SUBAPPLICATION Uebung_039a_AX (* Spiegelabfolge V2 mit Schrittkette *)
  (* Standard: 61499-2; Description: Copyright (c) 2023 Meisterschulen am Ostbahnhof This program and the accompanying materials are made available under the terms of the Eclipse Public License 2.0 which is available at https://www.eclipse.org/legal/epl-2.0/ SPDX-License-Identifier: EPL-2.0 *)
  (* Version 1.0, 2023-10-23, Franz Höpfinger, Meisterschulen am Ostbahnhof, initial API and implementation and/or initial documentation *)
  PACKAGE Uebungen;
  IMPORT isobus::UT::io::Softkey::SoftKeyActivationCode::SK_RELEASED;
  IMPORT Uebungen::const::UT::DefaultPool::SoftKey_F1;
  IMPORT Uebungen::const::UT::DefaultPool::SoftKey_F2;
  IMPORT Uebungen::const::UT::DefaultPool::SoftKey_F8;
  IMPORT Uebungen::const::UT::DefaultPool::OutputNumber_N1;
  IMPORT logiBUS::io::DI::logiBUS_DI::Input_I1;
  IMPORT logiBUS::io::DI::logiBUS_DI::Input_I2;
  IMPORT logiBUS::io::DI::logiBUS_DI::Input_I3;
  IMPORT logiBUS::io::DI::logiBUS_DI::Input_I4;
  IMPORT logiBUS::io::DI::logiBUS_DI_Events::BUTTON_SINGLE_CLICK;
  IMPORT logiBUS::io::DQ::logiBUS_DO::Output_Q1;
  IMPORT logiBUS::io::DQ::logiBUS_DO::Output_Q2;
  IMPORT logiBUS::utils::sequence::const::sequence::NO_TIME;
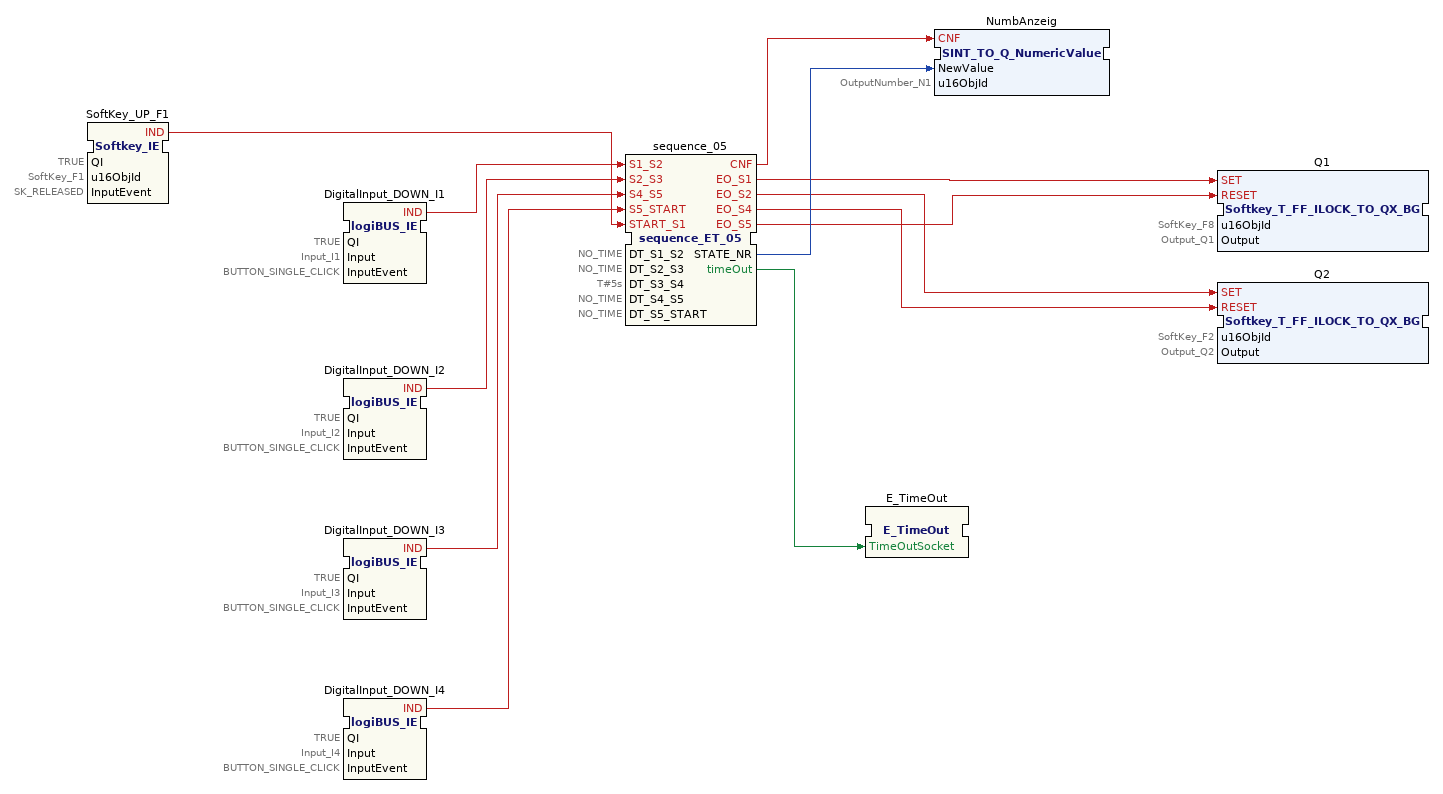
  FBS
    E_TimeOut : iec61499::events::E_TimeOut;
    DigitalInput_DOWN_I1 : logiBUS::io::DI::logiBUS_IE(QI := TRUE, Input := Input_I1, InputEvent := BUTTON_SINGLE_CLICK);
    DigitalInput_DOWN_I2 : logiBUS::io::DI::logiBUS_IE(QI := TRUE, Input := Input_I2, InputEvent := BUTTON_SINGLE_CLICK);
    DigitalInput_DOWN_I3 : logiBUS::io::DI::logiBUS_IE(QI := TRUE, Input := Input_I3, InputEvent := BUTTON_SINGLE_CLICK);
    DigitalInput_DOWN_I4 : logiBUS::io::DI::logiBUS_IE(QI := TRUE, Input := Input_I4, InputEvent := BUTTON_SINGLE_CLICK);
    sequence_05 : logiBUS::utils::sequence::combi::sequence_ET_05(DT_S1_S2 := NO_TIME, DT_S2_S3 := NO_TIME, DT_S3_S4 := T#5s, DT_S4_S5 := NO_TIME, DT_S5_START := NO_TIME);
    SoftKey_UP_F1 : isobus::UT::io::Softkey::Softkey_IE(QI := TRUE, u16ObjId := SoftKey_F1, InputEvent := SK_RELEASED);
  END_FBS
  SUBAPPS
    NumbAnzeig : MyLib::sys::SINT_TO_Q_NumericValue(u16ObjId := OutputNumber_N1);
    Q1 : MyLib::sys::Softkey_T_FF_ILOCK_TO_QX_BG(u16ObjId := SoftKey_F8, Output := Output_Q1);
    Q2 : MyLib::sys::Softkey_T_FF_ILOCK_TO_QX_BG(u16ObjId := SoftKey_F2, Output := Output_Q2);
  END_SUBAPPS
  EVENT_CONNECTIONS
    DigitalInput_DOWN_I1.IND TO sequence_05.S1_S2;
    DigitalInput_DOWN_I2.IND TO sequence_05.S2_S3;
    DigitalInput_DOWN_I3.IND TO sequence_05.S4_S5;
    DigitalInput_DOWN_I4.IND TO sequence_05.S5_START;
    sequence_05.CNF TO NumbAnzeig.CNF;
    SoftKey_UP_F1.IND TO sequence_05.START_S1;
    sequence_05.EO_S1 TO Q1.SET;
    sequence_05.EO_S2 TO Q2.SET;
    sequence_05.EO_S4 TO Q2.RESET;
    sequence_05.EO_S5 TO Q1.RESET;
  END_CONNECTIONS
  DATA_CONNECTIONS
    sequence_05.STATE_NR TO NumbAnzeig.NewValue;
  END_CONNECTIONS
  ADAPTER_CONNECTIONS
    sequence_05.timeOut TO E_TimeOut.TimeOutSocket;
  END_CONNECTIONS
END_SUBAPPLICATION
